# EPICS autosave request: iocBoot/iocVxWorks/auto_settings_SIS3801.req
file "SIS38XX_settings.req", P=$(P)
